FUNCTION_BLOCK FB_BaseImpulse IMPLEMENTS ITF_BaseImpulse
VAR
	tExitOn				: TON;
	tExitOff			: TON;
	rExitOn				: REAL;
	rExitOff			: REAL;
	
	bExecute			: BOOL;
	bFlashing			: BOOL;
	bExit				: BOOL;
	
END_VAR

THIS^.tExitOn 	(IN := (NOT THIS^.tExitOff.Q AND THIS^.bExecute AND THIS^.bFlashing),PT := REAL_TO_TIME (THIS^.rExitOn));
THIS^.tExitOff 	(IN := (THIS^.tExitOn.Q),PT := REAL_TO_TIME (THIS^.rExitOff));

THIS^.bExit		:= (NOT THIS^.tExitOn.Q AND THIS^.bFlashing) OR (THIS^.bExecute AND NOT THIS^.bFlashing);

METHOD PUBLIC GetExit : BOOL
VAR_INPUT
END_VAR
GetExit				:= THIS^.bExit;
END_METHOD

METHOD PUBLIC SetExecuteOff
VAR_INPUT
END_VAR
THIS^.bExecute				:= FALSE;
THIS^.bFlashing				:= FALSE;
END_METHOD

METHOD PUBLIC SetExecuteOn
VAR_INPUT
END_VAR
THIS^.bExecute			:= TRUE;
END_METHOD

METHOD PUBLIC SetFlashing
VAR_INPUT
	bIN				: BOOL;
END_VAR
THIS^.bFlashing				:= bIN;
END_METHOD

METHOD PUBLIC SetTimeOff
VAR_INPUT
	rIN: REAL;
END_VAR
THIS^.rExitOff			:= rIN;
END_METHOD

METHOD PUBLIC SetTimeOn
VAR_INPUT
	rIN					: REAL;
END_VAR
THIS^.rExitOn			:= rIN;
END_METHOD

END_FUNCTION_BLOCK

(* stored: Version 1.1.0.1
   POU FB_BaseImpulse: Id {6dbbd40b-fdc8-08db-2df3-88660c36c74c}, SpecialFunc None
   Method GetExit: Id {d6afa48a-7984-034a-072e-853ba8bb6126}
   Method SetExecuteOff: Id {7c2fc002-cb2b-0715-3606-95093d82e313}
   Method SetExecuteOn: Id {79ba7cd9-9e4c-05f2-24a5-31b5a2ae7391}
   Method SetFlashing: Id {dee2c5ed-cc5c-0510-1b11-5b7fc2649291}
   Method SetTimeOff: Id {206e5d9d-264a-000d-0e30-95795176ce5c}
   Method SetTimeOn: Id {140018c9-2914-0a4b-2ba2-7a795a2a66b7} *)
